{attribute addProperty BoxType "EK1122-0000-0018"}
{attribute addProperty Id "Beckhoff_ELM9xxxsub_EK1100EK1100_179A0949162"}
{attribute addProperty CRC "3758677293"}
{attribute addProperty SizeInBites "16"}
{attribute addProperty SizeInBytes "2"}
TYPE Beckhoff_ELM9xxxEK1122_E008DD2D EXTENDS EK1122_179A0949 :
STRUCT
	{attribute addProperty Name "Beckhoff_ELM9xxxsub_EK1100"}
	Beckhoff_ELM9xxxsub_EK1100 : EK1100_179A0949;
END_STRUCT
END_TYPE

(* stored: Version 1.2.0.0, ProductVersion 3.1.4024.9
   DUT Beckhoff_ELM9xxxEK1122_E008DD2D: Id {6101087a-6bdc-4161-bae1-df00e2d47cd1} *)
